FUNCTION F_ComputeUInt64Size : UDINT
VAR_INPUT
    anyUlint : ANY;
END_VAR
VAR
    nTmp   : ULINT;
END_VAR

memcpy(destAddr:= ADR(nTmp), srcAddr:= anyUlint.pValue, n:= MIN(TO_UDINT(anyUlint.diSize), SIZEOF(nTmp)));
F_ComputeUInt64Size := F_ComputeRawVarint64Size(nTmp);

END_FUNCTION

(* stored: Version 1.1.0.1
   POU F_ComputeUInt64Size: Id {bb4b8e0f-6024-456c-8b41-ca1717cde303}, SpecialFunc None *)
